(* CODESYS project SCADA-tankAndSortingPlant.export

Project tree, tasks and I/O mapping:
  Device : CODESYS Control Win V3 x64, CODESYS, version 3.5.22.30
    application Application
      libraries: Standard, 3.5.22.0 (System)
      task MainTask (cyclic, interval t#20ms, priority 1) calls PLC_PRG
      global variables FIO
      global variables SCADA
      function block FB_OperatorControl [ST]
      function block FB_PlantCoordinator [ST]
      function block FB_RackManager [ST]
      function block FB_Storage [ST]
      function block FB_Tank [ST]
      program PLC_PRG [ST]
      Symbols
      data type E_PlantState
      data type E_RackSlotState
      data type E_StorageState
      data type E_TankState
*)

// Device/Application/E_PlantState
{attribute 'qualified_only'}
{attribute 'strict'}
TYPE E_PlantState :
(
    CommittingInventory          := 60,
    DischargingBatch             := 40,
    Faulted                      := 900,
    Idle                         := 10,
    ReservingSlot                := 20,
    Stopped                      := 0,
    StoringProduct               := 50,
    WaitingForBatch              := 30,
    WaitingForStorageComplete    := 70
);
END_TYPE

// Device/Application/E_RackSlotState
{attribute 'qualified_only'}
{attribute 'strict'}
TYPE E_RackSlotState :
(
    Free      := 0,
    Occupied  := 20,
    Reserved  := 10,
    Unknown   := 900
);
END_TYPE

// Device/Application/E_StorageState
{attribute 'qualified_only'}
{attribute 'strict'}
TYPE E_StorageState :
(
    Complete                := 110,
    ExtendingToLoad         := 30,
    ExtendingToRack         := 70,
    Faulted                 := 900,
    Idle                    := 10,
    LiftingProduct          := 40,
    LoweringProduct         := 80,
    MovingToRack            := 60,
    ReceivingProduct        := 20,
    RetractingAfterDeposit  := 90,
    RetractingWithProduct   := 50,
    ReturningHome           := 100,
    Stopped                 := 0
);
END_TYPE

// Device/Application/E_TankState
{attribute 'qualified_only'}
{attribute 'strict'}
TYPE E_TankState :
(
    Stopped      := 0,
    Idle         := 10,
    Filling      := 20,
    BatchReady   := 30,
    Discharging  := 40,
    Faulted      := 100
);
END_TYPE

// Device/Application/FIO
{attribute 'qualified_only'}
VAR_GLOBAL
    // Operator-control commands and recovery status generated by the PLC
	xAutoRun: BOOL;
	xPlantEnable: BOOL;
	xPlantReset: BOOL;
	xRecoveryRequired: BOOL;
	
	// Factory I/O operator controls
	xAutoModeSelected: BOOL;
	
	// Factory I/O lifecycle feedback used for transaction recovery
	xFactoryIORunning: BOOL;
	
	// Released and healthy
	xEmergencyStopHealthy: BOOL;
	xResetPB: BOOL;
	xStartPB: BOOL;
	
	// Stop button not pressed
	xStopCircuitHealthy: BOOL;
	
	// Operator indication commands generated by the PLC
	xResetLightCmd: BOOL;
	xStartLightCmd: BOOL;
	xStopLightCmd: BOOL;

    // Tank and transfer feedback received from Factory I/O through Kepware
    rTankLevelV: REAL;
    xContainerAtFill: BOOL;
    xTankLevelHighHigh: BOOL;
	
	// Analog tank commands sent to Factory I/O
	rDischargeValveCmdV: REAL;
	rFillValveCmdV: REAL;
	
	// Boolean tank commands retained for diagnostics
	xDischargeValveCmd: BOOL;
	xFillValveCmd: BOOL;
	
	// Container supply command generated by the PLC
	xContainerEmitterCmd: BOOL;

    // Storage feedback received from Factory I/O
    xForkAtLeft: BOOL;
    xForkAtMiddle: BOOL;
    xForkAtRight: BOOL;
	xLoadBeamClear: BOOL;
    xMovingX: BOOL;
    xMovingZ: BOOL;

    // Storage actuator commands generated by the PLC
    wTargetPositionCmd: WORD := 55;
    xEntryConveyorCmd: BOOL;
    xForksLeftCmd: BOOL;
    xForksRightCmd: BOOL;
    xLiftCmd: BOOL;
    xLoadConveyorCmd: BOOL;
	
	(* 
		Commands for the four identical roller-conveyor sections
		Of Note (Learning) - 'ax' means an array of Bools 
	*)
	axRollerConveyorCmd: ARRAY[0..3] OF BOOL;

    // Public plant status and diagnostics
    ePlantState: E_PlantState := E_PlantState.Stopped;
    eStorageState: E_StorageState := E_StorageState.Stopped;
    eTankState: E_TankState := E_TankState.Stopped;
	xEmergencyActive: BOOL;
	xResetRequired: BOOL;
	
	// PLC-derived plant conditions
	xCraneAtHome: BOOL;
	xProductAtLoad: BOOL;
	xTransferPathClear: BOOL;
	
	(*
		Stack-light locations:
		[0] = infeed/emitter
		[1] = tank/filling position
		[2] = control panel
		[3] = outfeed/remover
	*)
	axStackGreenCmd: ARRAY[0..3] OF BOOL;
	axStackRedCmd: ARRAY[0..3] OF BOOL;
	axStackYellowCmd: ARRAY[0..3] OF BOOL;
	
	// Scaled tank measurement for control and diagnostics
	rTankLevelPct: REAL;

    uiFreeCount: UINT;
    uiOccupiedCount: UINT;
    uiReservedCount: UINT;
	uiUnknownCount: UINT;
	

    wReservedPosition: WORD;

    xDischargeTimeoutFault: BOOL;
    xFillTimeoutFault: BOOL;
    xHighHighFault: BOOL;
    xPlantFaulted: BOOL;
    xPlantRunning: BOOL;
    xRackFaulted: BOOL;
    xRackFull: BOOL;
    xSequenceFault: BOOL;
    xStepTimeoutFault: BOOL;
    xStorageFaulted: BOOL;
    xStorageReady: BOOL;
    xTankBatchReady: BOOL;
    xTankFaulted: BOOL;
    xWaitingForContainer: BOOL;
    xWaitingForStorage: BOOL;
END_VAR

// Device/Application/SCADA
{attribute 'qualified_only'}
VAR_GLOBAL
    // Momentary Ignition requests; cleared by the PLC after consumption
    xResetReq: BOOL;
    xStartReq: BOOL;
    xStopReq: BOOL;
END_VAR

// Device/Application/PLC_PRG
PROGRAM PLC_PRG
VAR
	//Comments retained for learning and reference points early on during learning

    // Plant control modules
	fbOperatorControl: FB_OperatorControl;
    fbPlantCoordinator: FB_PlantCoordinator;
    fbRackManager: FB_RackManager;
    fbStorage: FB_Storage;
    fbTank: FB_Tank;
	
	// Internal conveyor control
	iRollerConveyorIndex: INT;
	xTransferConveyorCmd: BOOL;
	
	//  Stack light warning devices display
	iStackLightIndex: INT;
	xStackGreenCmd: BOOL;
	xStackRedCmd: BOOL;
	xStackYellowCmd: BOOL;
END_VAR

(*
	The original warehouse sensor is normally true while its beam is clear.
	A product is present when the pallet interrupts that beam.
*)
FIO.xProductAtLoad := NOT FIO.xLoadBeamClear;

// Merge physical panel inputs with momentary SCADA requests
fbOperatorControl(
    xAutoModeSelected := FIO.xAutoModeSelected,
    xEmergencyStopHealthy := FIO.xEmergencyStopHealthy,
    xFactoryIORunning := FIO.xFactoryIORunning,
    xPlantFaulted := FIO.xPlantFaulted,
    xPlantRunning := FIO.xPlantRunning,
    xResetPB := FIO.xResetPB OR SCADA.xResetReq,
    xStartPB := FIO.xStartPB OR SCADA.xStartReq,
    xStopCircuitHealthy :=
        FIO.xStopCircuitHealthy
        AND NOT SCADA.xStopReq
);

// Acknowledge each request after FB_OperatorControl has evaluated it
SCADA.xResetReq := FALSE;
SCADA.xStartReq := FALSE;
SCADA.xStopReq := FALSE;

// Publish operator-control commands and diagnostics
FIO.xAutoRun := fbOperatorControl.xAutoRun;
FIO.xEmergencyActive := fbOperatorControl.xEmergencyActive;
FIO.xPlantEnable := fbOperatorControl.xEnable;
FIO.xPlantReset := fbOperatorControl.xReset;
FIO.xResetLightCmd := fbOperatorControl.xResetLightCmd;
FIO.xResetRequired := fbOperatorControl.xResetRequired;
FIO.xStartLightCmd := fbOperatorControl.xStartLightCmd;
FIO.xStopLightCmd := fbOperatorControl.xStopLightCmd;

(*
	Factory I/O starts the numerical crane at its known rest position.
	Position 55 is the commanded rest position; stopped movement and
	centred forks are used as the available home confirmation.
*)
FIO.xCraneAtHome :=
    (FIO.wTargetPositionCmd = 55)
    AND FIO.xForkAtMiddle
    AND NOT FIO.xMovingX
    AND NOT FIO.xMovingZ;

(*
	The v1 system permits only one product in material handling.
	The transfer path is available when storage is idle and its
	loading position does not already contain a product.
*)
FIO.xTransferPathClear :=
    fbStorage.xReady
    AND NOT FIO.xProductAtLoad;

(*
	The coordinator reads module status from the previous PLC scan
	and generates this scan's transaction commands
*)
fbPlantCoordinator(
    xAutoRun := FIO.xAutoRun,
	xEmergencyActive := FIO.xEmergencyActive,
    xEnable := FIO.xPlantEnable,
    xReset := FIO.xPlantReset,

    xContainerAtFill := FIO.xContainerAtFill,
    xTransferPathClear := FIO.xTransferPathClear,

    xRackCommitAck := fbRackManager.xCommitAck,
    xRackFaulted := fbRackManager.xFaulted,
    xRackFull := fbRackManager.xRackFull,
    xRackReservationValid := fbRackManager.xReservationValid,
    xRackReserveAck := fbRackManager.xReserveAck,

    xStorageDepositComplete := fbStorage.xDepositComplete,
    xStorageFaulted := fbStorage.xFaulted,
    xStorageReady := fbStorage.xReady,
    xStorageStoreComplete := fbStorage.xStoreComplete,

    xTankBatchReady := fbTank.xBatchReady,
    xTankDischargeComplete := fbTank.xDischargeComplete,
    xTankFaulted := fbTank.xFaulted,
    xTankReady := fbTank.xReady
);

// Rack inventory and reservation transactions
fbRackManager(
    xCommitRequest := fbPlantCoordinator.xRackCommitRequest,
    xEnable := fbPlantCoordinator.xModuleEnable,
	 xReservationMayBeOccupied :=
        fbPlantCoordinator.xReservationMayBeOccupied,
    xReserveRequest := fbPlantCoordinator.xRackReserveRequest,
    xReset := fbPlantCoordinator.xModuleReset
);

// Convert the Factory I/O 0–10 V level signal into 0–100%
FIO.rTankLevelPct := FIO.rTankLevelV * 10.0;

// Tank production module
fbTank(
    xEnable := fbPlantCoordinator.xModuleEnable,
    xDischargePermit := fbPlantCoordinator.xTankDischargePermit,
    xReset := fbPlantCoordinator.xModuleReset,
    xStartBatchReq := fbPlantCoordinator.xTankStartBatchReq,

    rLevelPct := FIO.rTankLevelPct,
    xLevelHighHigh := FIO.xTankLevelHighHigh,

    rEmptySetpointPct := 5.0,
    rFillSetpointPct := 80.0,
    tDischargeTimeout := T#2M,
    tFillTimeout := T#2M
);

// Automated storage module
fbStorage(
    xEnable := fbPlantCoordinator.xModuleEnable,
    xReset := fbPlantCoordinator.xModuleReset,
    xStoreRequest := fbPlantCoordinator.xStorageStoreRequest,

    xCraneAtHome := FIO.xCraneAtHome,
    xForkAtLeft := FIO.xForkAtLeft,
    xForkAtMiddle := FIO.xForkAtMiddle,
    xForkAtRight := FIO.xForkAtRight,
    xMovingX := FIO.xMovingX,
    xMovingZ := FIO.xMovingZ,
    xProductAtLoad := FIO.xProductAtLoad,

    wHomePosition := 55,
    xReservationValid := fbRackManager.xReservationValid,
    wReservedPosition := fbRackManager.wReservedPosition,

    tLiftTime := T#1500MS,
    tLowerTime := T#1500MS,
    tStepTimeout := T#2M
);

// Publish physical actuator commands through the external I/O boundary
FIO.xDischargeValveCmd := fbTank.xDischargeValveCmd;
FIO.xFillValveCmd := fbTank.xFillValveCmd;

// Convert the tank's Boolean valve commands into Factory I/O 0–10 V signals
IF fbTank.xDischargeValveCmd THEN
    FIO.rDischargeValveCmdV := 10.0;
ELSE
    FIO.rDischargeValveCmdV := 0.0;
END_IF;

IF fbTank.xFillValveCmd THEN
    FIO.rFillValveCmdV := 10.0;
ELSE
    FIO.rFillValveCmdV := 0.0;
END_IF;

// Request one empty container when the batch is ready for packaging
FIO.xContainerEmitterCmd := fbPlantCoordinator.xWaitingForContainer;

(*
    The transfer route has two valid movement requests:
    1. Bring an empty container to the filling position.
    2. Transfer the filled product towards storage.

    All four roller sections follow the same logical command.
	The loop distributes that command across the repeated equipment.
*)
xTransferConveyorCmd :=
    fbPlantCoordinator.xWaitingForContainer
    OR fbStorage.xEntryConveyorCmd;

FIO.xEntryConveyorCmd := xTransferConveyorCmd;

FOR iRollerConveyorIndex := 0 TO 3 DO
    FIO.axRollerConveyorCmd[iRollerConveyorIndex] :=
        xTransferConveyorCmd;
END_FOR;
FIO.xForksLeftCmd := fbStorage.xForksLeftCmd;
FIO.xForksRightCmd := fbStorage.xForksRightCmd;
FIO.xLiftCmd := fbStorage.xLiftCmd;
FIO.xLoadConveyorCmd := fbStorage.xLoadConveyorCmd;
FIO.wTargetPositionCmd := fbStorage.wTargetPositionCmd;

(*
    Stack-light priority:
    Red    = emergency, plant fault or interrupted recovery.
    Yellow = stopped, reset required or rack capacity unavailable.
    Green  = automatic production running normally.

    The conditions are mutually exclusive so only one colour
    is illuminated at a time.
*)
xStackRedCmd :=
    fbOperatorControl.xEmergencyActive
    OR fbPlantCoordinator.xFaulted
    OR fbPlantCoordinator.xRecoveryRequired;

xStackYellowCmd :=
    NOT xStackRedCmd
    AND (
        fbOperatorControl.xResetRequired
        OR fbRackManager.xRackFull
        OR NOT fbPlantCoordinator.xRunning
    );

xStackGreenCmd :=
    fbPlantCoordinator.xRunning
    AND NOT xStackRedCmd
    AND NOT xStackYellowCmd;

FOR iStackLightIndex := 0 TO 3 DO
    FIO.axStackGreenCmd[iStackLightIndex] := xStackGreenCmd;
    FIO.axStackRedCmd[iStackLightIndex] := xStackRedCmd;
    FIO.axStackYellowCmd[iStackLightIndex] := xStackYellowCmd;
END_FOR;

(*
	Final external-output interlock for the Factory I/O simulation.
	Numerical target zero stops the crane at its current position.
*)
IF fbOperatorControl.xEmergencyActive
    OR fbOperatorControl.xResetRequired
    OR fbPlantCoordinator.xFaulted
    OR fbPlantCoordinator.xRecoveryRequired
THEN
    FIO.rDischargeValveCmdV := 0.0;
    FIO.rFillValveCmdV := 0.0;
    FIO.wTargetPositionCmd := 0;

    FIO.xContainerEmitterCmd := FALSE;
    FIO.xDischargeValveCmd := FALSE;
    FIO.xEntryConveyorCmd := FALSE;
    FIO.xFillValveCmd := FALSE;
    FIO.xForksLeftCmd := FALSE;
    FIO.xForksRightCmd := FALSE;
    FIO.xLiftCmd := FALSE;
    FIO.xLoadConveyorCmd := FALSE;
	// Utilise the loop to control the multiple conveyors
    FOR iRollerConveyorIndex := 0 TO 3 DO
    FIO.axRollerConveyorCmd[iRollerConveyorIndex] := FALSE;
	END_FOR;
END_IF;

// Publish plant status and diagnostics
FIO.ePlantState := fbPlantCoordinator.eState;
FIO.eStorageState := fbStorage.eState;
FIO.eTankState := fbTank.eState;

FIO.uiFreeCount := fbRackManager.uiFreeCount;
FIO.uiOccupiedCount := fbRackManager.uiOccupiedCount;
FIO.uiReservedCount := fbRackManager.uiReservedCount;
FIO.uiUnknownCount := fbRackManager.uiUnknownCount;
FIO.wReservedPosition := fbRackManager.wReservedPosition;

FIO.xDischargeTimeoutFault := fbTank.xDischargeTimeoutFault;
FIO.xFillTimeoutFault := fbTank.xFillTimeoutFault;
FIO.xHighHighFault := fbTank.xHighHighFault;
FIO.xPlantFaulted := fbPlantCoordinator.xFaulted;
FIO.xPlantRunning := fbPlantCoordinator.xRunning;
FIO.xRackFaulted := fbRackManager.xFaulted;
FIO.xRackFull := fbRackManager.xRackFull;
FIO.xRecoveryRequired := fbPlantCoordinator.xRecoveryRequired;
FIO.xSequenceFault := fbPlantCoordinator.xSequenceFault;
FIO.xStepTimeoutFault := fbStorage.xStepTimeoutFault;
FIO.xStorageFaulted := fbStorage.xFaulted;
FIO.xStorageReady := fbStorage.xReady;
FIO.xTankBatchReady := fbTank.xBatchReady;
FIO.xTankFaulted := fbTank.xFaulted;
FIO.xWaitingForContainer := fbPlantCoordinator.xWaitingForContainer;
FIO.xWaitingForStorage := fbPlantCoordinator.xWaitingForStorage;

END_PROGRAM

// Device/Application/FB_OperatorControl
FUNCTION_BLOCK FB_OperatorControl
VAR_INPUT
	//Comments retained for learning and reference points early on during learning
	
    // Physical operator controls
    xAutoModeSelected: BOOL;
    xEmergencyStopHealthy: BOOL;
	xFactoryIORunning: BOOL;
    xPlantFaulted: BOOL;
	xPlantRunning: BOOL;
    xResetPB: BOOL;
    xStartPB: BOOL;
    xStopCircuitHealthy: BOOL;
END_VAR

VAR_OUTPUT
    // Commands and safety status supplied to the plant
    xAutoRun: BOOL;
    xEmergencyActive: BOOL;
    xEnable: BOOL;
    xReset: BOOL;
	xResetLightCmd: BOOL;
    xResetRequired: BOOL := TRUE;
	xStartLightCmd: BOOL;
    xStopLightCmd: BOOL;
END_VAR

VAR
    fbStartEdge: R_TRIG;
    xRunLatched: BOOL;
END_VAR

// Start is accepted only on a new button press
fbStartEdge(CLK := xStartPB);

(*
	Stopping OR resetting Factory I/O invalidates the current
	simulated transaction and requires operator acknowledgement. 
*)
IF NOT xFactoryIORunning THEN
    xResetRequired := TRUE;
    xRunLatched := FALSE;
END_IF;

// Emergency stop immediately removes the run request and requires reset
IF NOT xEmergencyStopHealthy THEN
    xResetRequired := TRUE;
    xRunLatched := FALSE;
END_IF;

// Normal stop conditions remove the run latch but do not create a fault
IF NOT xAutoModeSelected
    OR NOT xStopCircuitHealthy
    OR xPlantFaulted
THEN
    xRunLatched := FALSE;
END_IF;

// Reset is accepted only with healthy stop circuits and no run request
xReset :=
    xResetPB
    AND xEmergencyStopHealthy
	AND xFactoryIORunning
    AND xStopCircuitHealthy
    AND NOT xRunLatched;

// Reset and Start cannot be accepted during the same PLC scan
IF xReset THEN
    xResetRequired := FALSE;

ELSIF fbStartEdge.Q
    AND xAutoModeSelected
    AND xEmergencyStopHealthy
	AND xFactoryIORunning
    AND xStopCircuitHealthy
    AND NOT xPlantFaulted
    AND NOT xResetRequired
THEN
    xRunLatched := TRUE;
END_IF;

// Public operator-control outputs
xEmergencyActive := NOT xEmergencyStopHealthy;

xEnable :=
    xEmergencyStopHealthy
	AND xFactoryIORunning
    AND NOT xResetRequired;

xAutoRun :=
    xEnable
    AND xAutoModeSelected
    AND xRunLatched;
	
// Reset indication identifies a condition requiring operator acknowledgement
xResetLightCmd :=
    xResetRequired
    OR xPlantFaulted;

// Start indication reports actual plant activity
xStartLightCmd :=
    xEnable
    AND xPlantRunning
    AND NOT xPlantFaulted;

// Stop indication reports a healthy but stationary plant
xStopLightCmd :=
    xEnable
    AND NOT xPlantRunning
    AND NOT xPlantFaulted;

END_FUNCTION_BLOCK

// Device/Application/FB_PlantCoordinator
FUNCTION_BLOCK FB_PlantCoordinator
VAR_INPUT
	//Comments retained for learning and reference points early on during learning

    // Operator commands
    xAutoRun: BOOL;
	xEmergencyActive: BOOL;
    xEnable: BOOL;
    xReset: BOOL;

    // Filling and transfer sensors
    xContainerAtFill: BOOL;
    xTransferPathClear: BOOL;

    // Rack manager status
    xRackCommitAck: BOOL;
    xRackFaulted: BOOL;
    xRackFull: BOOL;
    xRackReservationValid: BOOL;
    xRackReserveAck: BOOL;

    // Storage module status
    xStorageDepositComplete: BOOL;
    xStorageFaulted: BOOL;
    xStorageReady: BOOL;
    xStorageStoreComplete: BOOL;

    // Tank module status
    xTankBatchReady: BOOL;
    xTankDischargeComplete: BOOL;
    xTankFaulted: BOOL;
    xTankReady: BOOL;
END_VAR

VAR_OUTPUT
    // Shared module control
    xModuleEnable: BOOL;
    xModuleReset: BOOL;

    // Rack manager commands
    xRackCommitRequest: BOOL;
    xRackReserveRequest: BOOL;

    // Storage module command
    xStorageStoreRequest: BOOL;

    // Tank module commands
    xTankDischargePermit: BOOL;
    xTankStartBatchReq: BOOL;

    // Plant status and diagnostics
    xFaulted: BOOL;
	xRecoveryRequired: BOOL;
    xRunning: BOOL;
    xSequenceFault: BOOL;
    xWaitingForContainer: BOOL;
    xWaitingForStorage: BOOL;
    eState: E_PlantState := E_PlantState.Stopped;
	
	// Rack recovery classification
    xReservationMayBeOccupied: BOOL;
END_VAR

VAR
    // Internal production-permission calculation
	xMaterialMayExistState: BOOL;
    xTankPrefillAllowed: BOOL;
END_VAR

(*
	Capture the transaction phase before fault handling can overwrite eState.
	From discharge onward, physical product may exist somewhere in the cell.
*)
xMaterialMayExistState :=
    (eState = E_PlantState.CommittingInventory) OR
    (eState = E_PlantState.DischargingBatch) OR
    (eState = E_PlantState.StoringProduct);

(*
    An emergency or loss of the Factory I/O lifecycle during an
    active transaction requires reservation recovery.
*)
IF (xEmergencyActive OR NOT xEnable)
    AND (eState <> E_PlantState.Stopped)
    AND (eState <> E_PlantState.Faulted)
THEN
    xRecoveryRequired := TRUE;
END_IF;

// Combine faults reported by the coordinator and plant modules
xFaulted :=
    xRackFaulted OR
	xRecoveryRequired OR
    xSequenceFault OR
    xStorageFaulted OR
    xTankFaulted;

// Reset is accepted only after automatic production has been stopped
IF xReset AND NOT xAutoRun THEN
	xRecoveryRequired := FALSE;
    xSequenceFault := FALSE;
    eState := E_PlantState.Stopped;
END_IF;

// Recalculate after a possible reset
xFaulted :=
    xRackFaulted OR
	xRecoveryRequired OR
    xSequenceFault OR
    xStorageFaulted OR
    xTankFaulted;

IF xFaulted THEN
    eState := E_PlantState.Faulted;
END_IF;

(* 
	Modules remain enabled while completing a controlled-stop transaction.
	In Stopped, a new AutoRun request is required before they are enabled,
	preventing Reset by itself from causing physical movement.
*)
xModuleEnable :=
    xEnable
    AND NOT xFaulted
    AND (
        xAutoRun
        OR (
            (eState <> E_PlantState.Faulted)
            AND (eState <> E_PlantState.Stopped)
        )
    );

xModuleReset := xReset AND NOT xAutoRun;

// Safe transaction-command defaults
xRackCommitRequest := FALSE;
xRackReserveRequest := FALSE;
xStorageStoreRequest := FALSE;
xTankDischargePermit := FALSE;
xTankStartBatchReq := FALSE;

// Default status values
xTankPrefillAllowed := FALSE;
xWaitingForContainer := FALSE;
xWaitingForStorage := FALSE;

IF xModuleEnable THEN

    CASE eState OF

        E_PlantState.Stopped:
            // AutoRun begins a new production transaction
            IF xAutoRun THEN
                eState := E_PlantState.Idle;
            END_IF;

        E_PlantState.Idle:
            // Do not begin another transaction after a controlled stop
            IF NOT xAutoRun THEN
                eState := E_PlantState.Stopped;

            // An unexpected existing reservation requires reconciliation
            ELSIF xRackReservationValid THEN
                xSequenceFault := TRUE;

            // RackFull blocks production but is not an equipment fault
            ELSIF NOT xRackFull THEN
                eState := E_PlantState.ReservingSlot;
            END_IF;

        E_PlantState.ReservingSlot:
            // Hold the request until the rack manager acknowledges it
            xRackReserveRequest := TRUE;

            IF xRackReserveAck THEN

                IF xRackReservationValid THEN
                    eState := E_PlantState.WaitingForBatch;

                ELSIF xRackFull THEN
                    eState := E_PlantState.Idle;

                ELSE
					(*
                    	An acknowledgement without a reservation or full rack
                    	indicates inconsistent transaction feedback
					*)
                    xSequenceFault := TRUE;
                END_IF;

            END_IF;

        E_PlantState.WaitingForBatch:
            IF NOT xRackReservationValid THEN
                xSequenceFault := TRUE;

            ELSIF xTankBatchReady THEN
                xWaitingForContainer := NOT xContainerAtFill;

                xWaitingForStorage :=
                    NOT xTransferPathClear OR
                    NOT xStorageReady;

                IF xContainerAtFill
                    AND xTransferPathClear
                    AND xStorageReady
                THEN
                    eState := E_PlantState.DischargingBatch;
                END_IF;
            END_IF;

        E_PlantState.DischargingBatch:
            // Permission remains active until the tank acknowledges completion
            xTankDischargePermit := TRUE;

            IF NOT xRackReservationValid THEN
                xSequenceFault := TRUE;

            ELSIF xTankDischargeComplete THEN
                eState := E_PlantState.StoringProduct;
            END_IF;

        E_PlantState.StoringProduct:
            // Storage owns the conveyor and crane sequence from this point
            xStorageStoreRequest := TRUE;

            IF NOT xRackReservationValid THEN
                xSequenceFault := TRUE;

            ELSIF xStorageDepositComplete THEN
                eState := E_PlantState.CommittingInventory;
            END_IF;

        E_PlantState.CommittingInventory:
            // The storage request remains active while inventory is committed
            xStorageStoreRequest := TRUE;
            xRackCommitRequest := TRUE;

            IF NOT xRackReservationValid
                AND NOT xRackCommitAck
            THEN
                xSequenceFault := TRUE;

            ELSIF xRackCommitAck THEN

                IF NOT xRackReservationValid THEN
                    eState :=
                        E_PlantState.WaitingForStorageComplete;
                ELSE
                    xSequenceFault := TRUE;
                END_IF;

            END_IF;

        E_PlantState.WaitingForStorageComplete:
            // The slot is occupied, but the crane must still return home
            xStorageStoreRequest := TRUE;

            IF xStorageStoreComplete THEN

                IF xAutoRun THEN
                    eState := E_PlantState.Idle;
                ELSE
                    eState := E_PlantState.Stopped;
                END_IF;

            END_IF;

        E_PlantState.Faulted:
            // Transaction commands remain at their safe defaults

    END_CASE;

END_IF;

// Start the batch allocated to the current transaction
xTankPrefillAllowed :=
    xModuleEnable
    AND xTankReady
    AND (eState = E_PlantState.WaitingForBatch);
(*
	While the crane handles the current case, prepare the next batch only
	when automatic production remains requested and another slot is free
*)
xTankPrefillAllowed :=
    xTankPrefillAllowed
    OR (
        xModuleEnable
        AND xAutoRun
        AND xTankReady
        AND NOT xRackFull
        AND (
            (eState = E_PlantState.StoringProduct) OR
            (eState = E_PlantState.CommittingInventory) OR
            (eState = E_PlantState.WaitingForStorageComplete)
        )
    );

xTankStartBatchReq := xTankPrefillAllowed;

xRunning :=
    xModuleEnable
    AND (eState <> E_PlantState.Stopped)
    AND (eState <> E_PlantState.Faulted);

// Recalculate after evaluating the sequence
xFaulted :=
    xRackFaulted OR
	xRecoveryRequired OR
    xSequenceFault OR
    xStorageFaulted OR
    xTankFaulted;
	
(* 
	Preserve whether the interrupted reservation might now represent
	physical material. RackManager uses this during Reset. 
*)
IF xFaulted
    AND xRackReservationValid
    AND xMaterialMayExistState
THEN
    xReservationMayBeOccupied := TRUE;
END_IF;
(*
	Clear the classification only after Reset has ended
	and reservation reconciliation has completed.
*)
IF NOT xReset
    AND (eState = E_PlantState.Stopped)
    AND NOT xRackReservationValid
THEN
    xReservationMayBeOccupied := FALSE;
END_IF;

// A newly detected fault removes every permission during this same scan
IF xFaulted THEN
    eState := E_PlantState.Faulted;
    xModuleEnable := FALSE;
    xRackCommitRequest := FALSE;
    xRackReserveRequest := FALSE;
    xStorageStoreRequest := FALSE;
    xTankDischargePermit := FALSE;
    xTankPrefillAllowed := FALSE;
    xTankStartBatchReq := FALSE;
    xWaitingForContainer := FALSE;
    xWaitingForStorage := FALSE;
    xRunning := FALSE;
END_IF;

END_FUNCTION_BLOCK

// Device/Application/FB_RackManager
FUNCTION_BLOCK FB_RackManager
VAR_INPUT
	//Comments retained for learning and reference points early on during learning

    // Commands from the plant coordinator
    xCommitRequest: BOOL;
    xEnable: BOOL;
	xReservationMayBeOccupied: BOOL;
    xReserveRequest: BOOL;
    xReset: BOOL;
END_VAR

VAR_OUTPUT
    // Rack inventory and calculated totals
    aSlotState: ARRAY[1..54] OF E_RackSlotState;
    uiFreeCount: UINT;
    uiOccupiedCount: UINT;
    uiReservedCount: UINT;
    uiUnknownCount: UINT;

    // Current reserved destination
    wReservedPosition: WORD;
    xReservationValid: BOOL;

    // Transaction acknowledgements
    xCommitAck: BOOL;
    xReserveAck: BOOL;

    // Module status and diagnostics
    xFaulted: BOOL;
    xRackFull: BOOL;
END_VAR

VAR
    // Internal control and slot-search variables
    iSlot: INT;
    wCandidatePosition: WORD;
	xInvalidOperationFault: BOOL;
END_VAR

// Acknowledgements remain high until their request returns low
IF NOT xCommitRequest THEN
    xCommitAck := FALSE;
END_IF;

IF NOT xReserveRequest THEN
    xReserveAck := FALSE;
END_IF;

(*
    Reset clears control faults only after all transaction requests
    have been removed.

    An unused pre-production reservation returns to Free.
    A reservation associated with possible physical material is
    quarantined as Unknown.
*)
IF xReset
    AND NOT xCommitRequest
    AND NOT xReserveRequest
THEN
    xInvalidOperationFault := FALSE;

    IF xReservationValid THEN

        IF (wReservedPosition >= 1)
            AND (wReservedPosition <= 54)
            AND (
                aSlotState[WORD_TO_INT(wReservedPosition)]
                = E_RackSlotState.Reserved
            )
        THEN

            IF xReservationMayBeOccupied THEN
                aSlotState[WORD_TO_INT(wReservedPosition)] :=
                    E_RackSlotState.Unknown;
            ELSE
                aSlotState[WORD_TO_INT(wReservedPosition)] :=
                    E_RackSlotState.Free;
            END_IF;

            wReservedPosition := 0;
            xReservationValid := FALSE;

        ELSE
            (*
                Retain the reservation information if its internal
                state is inconsistent, allowing investigation.
            *)
            xInvalidOperationFault := TRUE;
        END_IF;

    END_IF;

END_IF;

// Simultaneous transaction commands are invalid
IF xCommitRequest AND xReserveRequest THEN
    xInvalidOperationFault := TRUE;
END_IF;

xFaulted := xInvalidOperationFault;

IF xEnable AND NOT xFaulted THEN

    // Commit the currently reserved position as occupied
    IF xCommitRequest AND NOT xCommitAck THEN

        IF xReservationValid
            AND (wReservedPosition >= 1)
            AND (wReservedPosition <= 54)
            AND (
                aSlotState[WORD_TO_INT(wReservedPosition)]
                = E_RackSlotState.Reserved
            )
        THEN
            aSlotState[WORD_TO_INT(wReservedPosition)] :=
                E_RackSlotState.Occupied;

            xReservationValid := FALSE;
            wReservedPosition := 0;
            xCommitAck := TRUE;
        ELSE
            xInvalidOperationFault := TRUE;
        END_IF;

    // Select the first available rack position
    ELSIF xReserveRequest AND NOT xReserveAck THEN

        IF xReservationValid THEN
            // This v1 manager supports one active reservation
            xInvalidOperationFault := TRUE;
        ELSE
            wCandidatePosition := 0;
            wReservedPosition := 0;

            FOR iSlot := 1 TO 54 DO

                IF (wCandidatePosition = 0)
                    AND (
                        aSlotState[iSlot]
                        = E_RackSlotState.Free
                    )
                THEN
                    wCandidatePosition := INT_TO_WORD(iSlot);
                END_IF;

            END_FOR;

            IF wCandidatePosition <> 0 THEN
                aSlotState[WORD_TO_INT(wCandidatePosition)] :=
                    E_RackSlotState.Reserved;

                wReservedPosition := wCandidatePosition;
                xReservationValid := TRUE;
            END_IF;

            // Acknowledge even when full; validity reports the outcome
            xReserveAck := TRUE;
        END_IF;

    END_IF;

END_IF;

// Recalculate inventory totals every scan
uiFreeCount := 0;
uiOccupiedCount := 0;
uiReservedCount := 0;
uiUnknownCount := 0;

FOR iSlot := 1 TO 54 DO

    CASE aSlotState[iSlot] OF

        E_RackSlotState.Free:
            uiFreeCount := uiFreeCount + 1;

        E_RackSlotState.Occupied:
            uiOccupiedCount := uiOccupiedCount + 1;

        E_RackSlotState.Reserved:
            uiReservedCount := uiReservedCount + 1;

        E_RackSlotState.Unknown:
            uiUnknownCount := uiUnknownCount + 1;

    END_CASE;

END_FOR;

xRackFull := uiFreeCount = 0;
xFaulted := xInvalidOperationFault;

END_FUNCTION_BLOCK

// Device/Application/FB_Storage
FUNCTION_BLOCK FB_Storage
VAR_INPUT
	//Comments retained for learning and reference points early on during learning

    // Commands from the plant coordinator
    xEnable: BOOL;
	xReset: BOOL;
    xStoreRequest: BOOL;
    
    // Product and crane feedback
	xCraneAtHome: BOOL;
    xForkAtLeft: BOOL;
    xForkAtMiddle: BOOL;
    xForkAtRight: BOOL;
    xMovingX: BOOL;
    xMovingZ: BOOL;
	xProductAtLoad: BOOL;

    // Reserved destination supplied by the rack manager
	wHomePosition: WORD := 55;
    xReservationValid: BOOL;
    wReservedPosition: WORD;
	

    // Adjustable timing limits
	tLiftTime: TIME := T#2S;
    tLowerTime: TIME := T#2s;
    tStepTimeout: TIME := T#30s;
END_VAR

VAR_OUTPUT
    // Crane and conveyor commands
    xEntryConveyorCmd: BOOL;
    xLoadConveyorCmd: BOOL;
    xForksLeftCmd: BOOL;
    xForksRightCmd: BOOL;
    xLiftCmd: BOOL;
    wTargetPositionCmd: WORD := 55;

    // Module status
	xDepositComplete: BOOL;
	xFaulted: BOOL;
	xReady: BOOL;
    xStoreComplete: BOOL;
    xStepTimeoutFault: BOOL;
    eState: E_StorageState := E_StorageState.Stopped;
END_VAR

VAR
    ePreviousState: E_StorageState := E_StorageState.Stopped;
    fbLiftTimer: TON;
    fbLowerTimer: TON;
    fbStepTimeout: TON;
	wActivePosition: WORD;
    xCommandArmed: BOOL;
    xMotionStarted: BOOL;
	xReservationFault: BOOL;
    xStateChanged: BOOL;
    xTimedStep: BOOL;
END_VAR

// Timers used for vertical movements without direct position feedback
fbLiftTimer(
    IN := xEnable AND (eState = E_StorageState.LiftingProduct),
    PT := tLiftTime
);

fbLowerTimer(
    IN := xEnable AND (eState = E_StorageState.LoweringProduct),
    PT := tLowerTime
);

// Establish current fault status
xFaulted :=
    xReservationFault OR
    xStepTimeoutFault;
	
(*
	Reset clears control faults and returns the sequence
	to a non-moving baseline.
	Rack inventory is owned separately by FB_RackManager.
*)
IF xReset THEN
    eState := E_StorageState.Stopped;
    wActivePosition := 0;
    wTargetPositionCmd := 0;

    xDepositComplete := FALSE;
    xMotionStarted := FALSE;
    xReservationFault := FALSE;
    xStepTimeoutFault := FALSE;
END_IF;

// Recalculate after a possible reset
xFaulted :=
    xReservationFault OR
    xStepTimeoutFault;

IF xFaulted THEN
    eState := E_StorageState.Faulted;
END_IF;

// A request must return low before another transaction is accepted
IF xReset OR xFaulted THEN
    xCommandArmed := FALSE;
ELSIF NOT xStoreRequest THEN
    xCommandArmed := TRUE;
END_IF;

// Safe Boolean output defaults
xEntryConveyorCmd := FALSE;
xLoadConveyorCmd := FALSE;
xForksLeftCmd := FALSE;
xForksRightCmd := FALSE;
xLiftCmd := FALSE;
xReady := FALSE;
xStoreComplete := FALSE;

IF xEnable
		AND NOT xFaulted
		AND NOT xReset
	THEN

    CASE eState OF

        E_StorageState.Stopped:
            IF xCraneAtHome AND xForkAtMiddle THEN
                eState := E_StorageState.Idle;
            ELSE
                wTargetPositionCmd := wHomePosition;
                xMotionStarted := FALSE;
                eState := E_StorageState.ReturningHome;
            END_IF;

        E_StorageState.Idle:
            wTargetPositionCmd := wHomePosition;

            IF xStoreRequest AND xCommandArmed THEN

                IF xReservationValid
                    AND (wReservedPosition >= 1)
                    AND (wReservedPosition <= 54)
                THEN
                    wActivePosition := wReservedPosition;
                    xDepositComplete := FALSE;
                    xCommandArmed := FALSE;
                    eState := E_StorageState.ReceivingProduct;
                ELSE
                    xReservationFault := TRUE;
                END_IF;

            END_IF;

        E_StorageState.ReceivingProduct:
            IF xProductAtLoad THEN
                eState := E_StorageState.ExtendingToLoad;
            ELSE
                xEntryConveyorCmd := TRUE;
                xLoadConveyorCmd := TRUE;
            END_IF;

        E_StorageState.ExtendingToLoad:
            xForksLeftCmd := TRUE;

            IF xForkAtLeft THEN
                eState := E_StorageState.LiftingProduct;
            END_IF;

        E_StorageState.LiftingProduct:
            xForksLeftCmd := TRUE;
            xLiftCmd := TRUE;

            IF fbLiftTimer.Q THEN
                eState := E_StorageState.RetractingWithProduct;
            END_IF;

        E_StorageState.RetractingWithProduct:
            xLiftCmd := TRUE;

            IF xForkAtMiddle THEN
                xMotionStarted := FALSE;
                eState := E_StorageState.MovingToRack;
            END_IF;

        E_StorageState.MovingToRack:
            xLiftCmd := TRUE;
            wTargetPositionCmd := wActivePosition;

            IF xMovingX OR xMovingZ THEN
                xMotionStarted := TRUE;
            END_IF;

            IF xMotionStarted
                AND NOT xMovingX
                AND NOT xMovingZ
            THEN
                xMotionStarted := FALSE;
                eState := E_StorageState.ExtendingToRack;
            END_IF;

        E_StorageState.ExtendingToRack:
            xLiftCmd := TRUE;
            xForksRightCmd := TRUE;
            wTargetPositionCmd := wActivePosition;

            IF xForkAtRight THEN
                eState := E_StorageState.LoweringProduct;
            END_IF;

        E_StorageState.LoweringProduct:
            xForksRightCmd := TRUE;
            wTargetPositionCmd := wActivePosition;

            IF fbLowerTimer.Q THEN
                eState := E_StorageState.RetractingAfterDeposit;
            END_IF;

        E_StorageState.RetractingAfterDeposit:
            wTargetPositionCmd := wActivePosition;

            IF xForkAtMiddle THEN
                // Inventory may now be committed by the rack manager
                xDepositComplete := TRUE;
                xMotionStarted := FALSE;
                eState := E_StorageState.ReturningHome;
            END_IF;

        E_StorageState.ReturningHome:
            wTargetPositionCmd := wHomePosition;

            IF xMovingX OR xMovingZ THEN
                xMotionStarted := TRUE;
            END_IF;

            IF xForkAtMiddle
                AND (
                    xCraneAtHome
                    OR (
                        xMotionStarted
                        AND NOT xMovingX
                        AND NOT xMovingZ
                    )
                )
            THEN
                xMotionStarted := FALSE;

                IF xDepositComplete THEN
                    eState := E_StorageState.Complete;
                ELSE
                    // Startup or fault-recovery homing
                    eState := E_StorageState.Idle;
                END_IF;
            END_IF;

        E_StorageState.Complete:
            wTargetPositionCmd := wHomePosition;
            xStoreComplete := TRUE;

            // Hold completion until the coordinator removes its request
            IF NOT xStoreRequest THEN
                xDepositComplete := FALSE;
                xStoreComplete := FALSE;
                wActivePosition := 0;
                eState := E_StorageState.Idle;
            END_IF;

        E_StorageState.Faulted:
            // Boolean commands remain at their safe defaults

    END_CASE;

END_IF;

// States which must make progress within the configured timeout
xTimedStep :=
    (eState = E_StorageState.ReceivingProduct) OR
    (eState = E_StorageState.ExtendingToLoad) OR
    (eState = E_StorageState.LiftingProduct) OR
    (eState = E_StorageState.RetractingWithProduct) OR
    (eState = E_StorageState.MovingToRack) OR
    (eState = E_StorageState.ExtendingToRack) OR
    (eState = E_StorageState.LoweringProduct) OR
    (eState = E_StorageState.RetractingAfterDeposit) OR
    (eState = E_StorageState.ReturningHome);

// Reset the common timer for one scan whenever the state changes
xStateChanged := eState <> ePreviousState;

fbStepTimeout(
    IN := xEnable AND xTimedStep AND NOT xStateChanged,
    PT := tStepTimeout
);

ePreviousState := eState;

IF fbStepTimeout.Q THEN
    xStepTimeoutFault := TRUE;
END_IF;

// Recalculate after timeout evaluation
xFaulted :=
    xReservationFault OR
    xStepTimeoutFault;

// A newly detected fault stops all movement commands immediately
IF xFaulted THEN
    eState := E_StorageState.Faulted;
	wTargetPositionCmd := 0;
    xEntryConveyorCmd := FALSE;
    xLoadConveyorCmd := FALSE;
    xForksLeftCmd := FALSE;
    xForksRightCmd := FALSE;
    xLiftCmd := FALSE;
    xCommandArmed := FALSE;
END_IF;

// Public module status
xReady :=
    xEnable
    AND NOT xFaulted
    AND (eState = E_StorageState.Idle);

END_FUNCTION_BLOCK

// Device/Application/FB_Tank
FUNCTION_BLOCK FB_Tank
VAR_INPUT
	//Comments retained for learning and reference points early on during learning	

    // Commands and permissions from the plant coordinator
    xEnable: BOOL;
	xDischargePermit: BOOL;
    xReset: BOOL;
    xStartBatchReq: BOOL;

    // Physical tank measurements
    rLevelPct: REAL;
    xLevelHighHigh: BOOL;

    // Adjustable process settings
	rEmptySetpointPct:REAL := 5.0;
    rFillSetpointPct: REAL := 80.0;
	tDischargeTimeout: TIME := T#20S;
    tFillTimeout: TIME := T#30S;
END_VAR

VAR_OUTPUT
    // Commands sent towards physical actuators
	xDischargeValveCmd: BOOL;
    xFillValveCmd: BOOL;

    // Status reported to the plant coordinator
    xBatchReady: BOOL;
	xDischargeComplete: BOOL;
	xFaulted: BOOL;
	xReady: BOOL;

    // Individual fault diagnostics
	xDischargeTimeoutFault: BOOL;
	xFillTimeoutFault: BOOL;
    xHighHighFault: BOOL;
    

    // Current state for diagnostics and visualization
    eState: E_TankState := E_TankState.Stopped;
END_VAR

VAR
    // Private timer instances
	fbDischargeTimeout: TON;
    fbFillTimeout: TON;
	xCommandArmed: BOOL;
	xTankEmpty: BOOL;
END_VAR

// Convert the analog reading into a reusable tank status
xTankEmpty := rLevelPct <= rEmptySetpointPct;

// High-high is a trip: even a brief sensor signal remains latched
IF xLevelHighHigh THEN
    xHighHighFault := TRUE;
END_IF;

// Establish the current combined fault status
xFaulted :=
    xHighHighFault OR
    xFillTimeoutFault OR
    xDischargeTimeoutFault;

(*
	Reset returns both faulted and interrupted tank sequences
	to a known non-moving baseline.
	A live high-high condition prevents fault clearance.
*)
IF xReset AND NOT xLevelHighHigh THEN
    eState := E_TankState.Stopped;

    xHighHighFault := FALSE;
    xFillTimeoutFault := FALSE;
    xDischargeTimeoutFault := FALSE;
END_IF;

// Recalculate after a possible reset
xFaulted :=
    xHighHighFault OR
    xFillTimeoutFault OR
    xDischargeTimeoutFault;

IF xFaulted THEN
    eState := E_TankState.Faulted;
END_IF;

// Requests must return low after startup, reset or fault
IF xReset OR xFaulted THEN
    xCommandArmed := FALSE;
ELSIF NOT xStartBatchReq AND NOT xDischargePermit THEN
    xCommandArmed := TRUE;
END_IF;

// Hold completion until the coordinator removes its discharge permit
IF xReset OR xFaulted OR NOT xDischargePermit THEN
    xDischargeComplete := FALSE;
END_IF;

// Safe actuator defaults for every scan
xFillValveCmd := FALSE;
xDischargeValveCmd := FALSE;

IF xEnable
		AND NOT xFaulted
		AND NOT xReset
	THEN

    CASE eState OF

        E_TankState.Stopped:
			// Determine a safe starting state from the physical level
			IF rLevelPct >= rFillSetpointPct THEN
				eState := E_TankState.BatchReady;
			ELSE
				eState := E_TankState.Idle;
			END_IF;

        E_TankState.Idle:
            IF xStartBatchReq AND xCommandArmed THEN
                eState := E_TankState.Filling;
                xCommandArmed := FALSE;
            END_IF;

        E_TankState.Filling:
            IF rLevelPct >= rFillSetpointPct THEN
                eState := E_TankState.BatchReady;
            ELSE
                xFillValveCmd := TRUE;
            END_IF;

        E_TankState.BatchReady:
            IF xDischargePermit AND xCommandArmed THEN
                eState := E_TankState.Discharging;
                xCommandArmed := FALSE;
            END_IF;

        E_TankState.Discharging:
			IF xTankEmpty THEN
				xDischargeComplete := TRUE;
				eState := E_TankState.Idle;
		
			ELSIF xDischargePermit THEN
				xDischargeValveCmd := TRUE;
			END_IF;

        E_TankState.Faulted:
			xFillValveCmd := FALSE;
			xDischargeValveCmd := FALSE;

    END_CASE;

END_IF;

// Time spent in each active process state
fbFillTimeout(
    IN := xEnable AND (eState = E_TankState.Filling),
    PT := tFillTimeout
);

fbDischargeTimeout(
    IN := xEnable AND (eState = E_TankState.Discharging),
    PT := tDischargeTimeout
);

// Latch timeout faults
IF fbFillTimeout.Q THEN
    xFillTimeoutFault := TRUE;
END_IF;

IF fbDischargeTimeout.Q THEN
    xDischargeTimeoutFault := TRUE;
END_IF;

// Recalculate after evaluating the timers
xFaulted :=
    xHighHighFault OR
    xFillTimeoutFault OR
    xDischargeTimeoutFault;

// A newly detected fault closes both valves during this same scan
IF xFaulted THEN
    eState := E_TankState.Faulted;
    xFillValveCmd := FALSE;
    xDischargeValveCmd := FALSE;
    xCommandArmed := FALSE;
	xDischargeComplete := FALSE;
END_IF;

// Final defensive interlock: filling and discharge can never coexist
IF xFillValveCmd AND xDischargeValveCmd THEN
    xFillValveCmd := FALSE;
    xDischargeValveCmd := FALSE;
END_IF;

// Externally visible state information
xBatchReady := eState = E_TankState.BatchReady;
xReady :=
    xEnable
    AND NOT xFaulted
    AND xCommandArmed
    AND (eState = E_TankState.Idle);

END_FUNCTION_BLOCK
